FUNCTION_BLOCK FB_DataStuff

VAR
	// The array of data for each instance of FB_DataStuff
	a2dArray : ARRAY[1..1000] OF ARRAY[1..3] OF STRING;
	
	// The value that will be referenced to and calculated amongst the runners
	nValueToCalculate : UINT := 100;
	
	// This will keep track of the index in which the mStoreData method will place data in
	nIndexCounter : UINT := 0;
END_VAR

// Check if nIndexCounter is below the size of the objects array
IF nIndexCounter < 1000 THEN
	// Increment nIndexCounter by 1, to place in the next index of objects array
	nIndexCounter := nIndexCounter + 1;
	
	// Call mRunnerOne method
	mRunnerOne(pDataTable := a2dArray, // Send it the objects array
			   nIndexLocation := nIndexCounter, // Send the current index to be placed in
			   nRunnerValue := nValueToCalculate); // Send the objects nRunnerValue to calculate
	// ^^ Inside the method, it will create the references to the original array of the object
	//		rather than just creating a copy of it
			
	// Increment nIndexCounter by 1, to place in the next index of objects array   
	nIndexCounter := nIndexCounter + 1;
	
	// Call mRunnerOne method
	mRunnerTwo(pDataTable := a2dArray,  // Send it the objects array 
			   nIndexLocation := nIndexCounter,// Send the current index to be placed in
			   nRunnerValue := nValueToCalculate); // Send the objects nRunnerValue to calculate
	// ^^ Inside the method, it will create the references to the original array of the object
	//		rather than just creating a copy of it
END_IF

METHOD mRunnerOne : BOOL

VAR_INPUT
	// Create an array that references the objects array 
	pDataTable : REFERENCE TO ARRAY[1..1000] OF ARRAY[1..3] OF STRING;
	
	// This was sent, and will be forwarded to the following save function
	nIndexLocation : UINT;
	
	// Create a reference UINT of the objects value to calculate
	//    this way, both can edit the original variable at the same time
	nRunnerValue : REFERENCE TO UINT;
END_VAR

VAR
	// Local variable to send to the following save function, to ID that this is the sender
	nThisRunner : UINT := 1;
END_VAR
// Make the calculation that this runner is responsible for, 
//    and set it directly to the objects nValueToCalculate
nRunnerValue := nRunnerValue + 1;

// Call the mStoreData method to store the current entry that this runner calculated
//   after the subsequent nRunnerValue updated the objects nValueToCalculate data
//   this could mean that the data being stored could be old if the other runner 
//   updates the reference value
mStoreData(pDataTableOp := pDataTable, // Send the method the referenced table, which it will reference too
		   nIndexToStoreIn := nIndexLocation, // Send the index passed from the FB for tracking purposes
		   nValue := nRunnerValue, // Send it the referenced nRunnerValue  NOTE A*
		   nRunnerNumber := nThisRunner);
		   
// NOTE A: It is noteworthy that it is sending the referenced value of the nRunnerValue
//   instead of the result that the runner came to inside this method. 
//   That means that if the referenced nRunnerValue was changed by another runner between
//   the time that this runner calculated, and then stored; the mStoreData function would
//   then receive the most up to data value (from the other runner that was able to save
//   before this could call the save), rather than the value that this runner calculated.
//   - If the value of what this runner calculated was desired instead, then passing it
//   by value would be a better alternative. Which would be done by creating a local variable
//   and setting the calculation equal to that, and sending that value to the mStoreData. 
//   - Thus having multiple runners making calculations and updating the variable directly 
//   by reference has risks and race conditions if there was a slight delay with a runner
//   leading to their calculations and stores out of sync.
END_METHOD

METHOD mRunnerTwo : BOOL

VAR_INPUT
	// Create an array that references the objects array 
	pDataTable : REFERENCE TO ARRAY[1..1000] OF ARRAY[1..3] OF STRING;
	
	// This was sent, and will be forwarded to the following save function
	nIndexLocation : UINT;
	
	// Create a reference UINT of the objects value to calculate
	//    this way, both can edit the original variable at the same time
	nRunnerValue : REFERENCE TO UINT;
END_VAR

VAR
	// Local variable to send to the following save function, to ID that this is the sender
	nThisRunner : UINT := 2;
END_VAR
// Make the calculation that this runner is responsible for, 
//    and set it directly to the objects nValueToCalculate
nRunnerValue := nRunnerValue - 1;

// Call the mStoreData method to store the current entry that this runner calculated
//   after the subsequent nRunnerValue updated the objects nValueToCalculate data
//   this could mean that the data being stored could be old if the other runner 
//   updates the reference value
mStoreData(pDataTableOp := pDataTable, // Send the method the referenced table, which it will reference too
		   nIndexToStoreIn := nIndexLocation, // Send the index passed from the FB for tracking purposes
		   nValue := nRunnerValue, // Send it the referenced nRunnerValue  NOTE A*
		   nRunnerNumber := nThisRunner);
		   
// NOTE A: It is noteworthy that it is sending the referenced value of the nRunnerValue
//   instead of the result that the runner came to inside this method. 
//   That means that if the referenced nRunnerValue was changed by another runner between
//   the time that this runner calculated, and then stored; the mStoreData function would
//   then receive the most up to data value (from the other runner that was able to save
//   before this could call the save), rather than the value that this runner calculated.
//   - If the value of what this runner calculated was desired instead, then passing it
//   by value would be a better alternative. Which would be done by creating a local variable
//   and setting the calculation equal to that, and sending that value to the mStoreData. 
//   - Thus having multiple runners making calculations and updating the variable directly 
//   by reference has risks and race conditions if there was a slight delay with a runner
//   leading to their calculations and stores out of sync.
END_METHOD

METHOD mStoreData : BOOL

VAR_INPUT
	// Create the final reference to the original array in the object
	pDataTableOp : REFERENCE TO ARRAY[1..1000] OF ARRAY[1..3] OF STRING;
	
	// Receive the index to store, passed down from FB_DataStuff -> mRunner(number) -> here
	nIndexToStoreIn : UINT;
	
	// Receive the nValue from the latest reference to the nValueToCalculate from FB_DataStuff
	//  the reference chain is FB_DataStuff -> mRunner(number) 
	//  Note that the reference chain doesn't go to -> here, see NOTE A in mRunnerOne or mRunnerTwo
	nValue : UINT; 
	
	// Variable passed by the mRunner(number) that is calling, to ID the caller in the array
	nRunnerNumber : UINT;
END_VAR

VAR
	// Strings that will convert the incoming UINTs into STRINGS to be stored in array : STRING
	sCurrentStringA : STRING;
	sCurrentStringB : STRING;
END_VAR
// Convert the input values from the caller to STRING to be stored into array
sCurrentStringA := UINT_TO_STRING(nValue);
sCurrentStringB := UINT_TO_STRING(nRunnerNumber);

// pDataTable is referenced from FB_DataStuff -> mRunner(number) -> here
// This is so the array in the function block is updated directly from this function
pDataTableOp[nIndexToStoreIn][1] := sCurrentStringA;
pDataTableOp[nIndexToStoreIn][2] := sCurrentStringB;

// NOTE B: Although the scope of this exercise allows for just calling the array directly in 
//   the FB_DataStuff since it is an instance of an object and that data is linked to the instance
//   this is still relevant when passing to data to other Function Blocks (Classes), Methods, or
//   Functions outside the scope of this Function Block. It also demonstrates that you can 
//   chain a reference through multiple functions so that the lowest level method can still 
//   make a direct change to the highest level scope of the program, or in a scope that is 
//   within other FB's, Methods, or Functions.
//   - This is useful for data types that are massive in size, which would lead to passing
//   by value taking longer to copy the data over to another local variable; this is not
//   only time consuming, but it is also memory consuming as passing by value essentially 
//   doubles the amount of memory being allocated for the same data type. So in the interest
//   of saving time and space, it could benefit to pass by reference rather than value.
//   - The risks associated with this is race conditions, where two methods are working on 
//   the same data and may interupt eachothers results by changing the original value, 
//   leading to unexpected outcomes for data results. So caution should be exercised when
//   having multiple methods editing the same referenced value in separate places, especially
//   in TwinCAT where they can run parallel. 
//   - The secondary risk associated with it is that, since the method is directly affecting
//   the original copy of the data, if an error occurs and say it overwrites the data for a log,
//   then the original copy of the data is overwritten and thus lost. So the two scenarios
//   of preserving time and space, plus protecting the original copy of that data are to be 
//   considered when working with references. The same applies to pointers.
END_METHOD

END_FUNCTION_BLOCK

(* stored: Version 1.1.0.1, ProductVersion 3.1.4024.12
   POU FB_DataStuff: Id {5de43432-b6a0-4bfd-a085-0227690ebfb9}, SpecialFunc None
   Method mRunnerOne: Id {4c35da92-dbaa-462a-b449-f72ec02b6747}
   Method mRunnerTwo: Id {017cb03a-c4b4-4fa7-be8a-82cf29a99e89}
   Method mStoreData: Id {7643b4a4-143b-4065-9533-062b0b195bbd} *)
